SUBAPPLICATION Uebung_000_AX (* Einfache Addition *)
  (* Standard: 61499-2; Description: Copyright (c) 2023 Meisterschulen am Ostbahnhof This program and the accompanying materials are made available under the terms of the Eclipse Public License 2.0 which is available at https://www.eclipse.org/legal/epl-2.0/ SPDX-License-Identifier: EPL-2.0 *)
  (* Version 1.0, 2026-01-16, Franz Höpfinger, Meisterschulen am Ostbahnhof, initial API and implementation and/or initial documentation *)
  PACKAGE Uebungen;
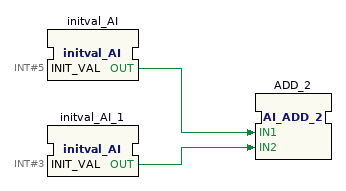
  FBS
    ADD_2 : adapter::iec61131::arithmetic::AI_ADD_2;
    initval_AI : adapter::types::unidirectional::AI::initval::initval_AI(INIT_VAL := INT#5);
    initval_AI_1 : adapter::types::unidirectional::AI::initval::initval_AI(INIT_VAL := INT#3);
  END_FBS
  ADAPTER_CONNECTIONS
    initval_AI.OUT TO ADD_2.IN1;
    initval_AI_1.OUT TO ADD_2.IN2;
  END_CONNECTIONS
END_SUBAPPLICATION
